PROGRAM MAIN
VAR
	nNum : DINT := 60000;
	fbMotor1 : FB_Motor ;
	fbMotor2 : FB_Motor ;
	
	fbTata : FB_TataNexon ;
	fbCar : POINTER TO FB_Car;
	
	iVehicle : I_Vehicle;
	pPoint1 : POINTER TO I_Vehicle;
	bRun: BOOL;
	num : INT;
	bCopyStart : BOOL;
END_VAR
VAR PERSISTENT
	num2 : INT := 323;
END_VAR
VAR CONSTANT
	num3 : INT := 34;
END_VAR

IF bRun THEN
	fbMotor1.Start();
	fbMotor1.Start();
	num := fbMotor1.nNum;
	fbMotor1.nNum := 433;
	bCopyStart := fbMotor1.bStart;
	bRun := FALSE;
END_IF
IF TRANS1 THEN
	//fbCar^.Running();
	fbTata();
END_IF
iVehicle := fbTata;
pPoint1 := ADR(iVehicle);

pPoint1^.Drive();

TRANSITION TRANS1:
TRANS1 := TRUE;
END_TRANSITION

END_PROGRAM

(* stored: Version 1.1.0.1, ProductVersion 3.1.4024.16
   POU MAIN: Id {e2595925-248a-4933-8312-1c95a489eb32}, SpecialFunc None
   Transition TRANS1: Id {11ed6e56-be5d-4a05-a3e9-39991f5af975} *)
